# EPICS substitutions: db/elveFlow.substitutions
# asyn record
file "$(ASYN)/db/asynRecord.db"
{
pattern
{ P,	 		    R, 	  PORT,        ADDR, IMAX, OMAX}
{"XF11ID-ES\{elveFlowOB1\}:", asyn, elveFlowOB1, 0,    80,   80}
}
# Analog outputs, analog inputs
file "$(ELVEFLOW)/db/elveFlow.template"
{
pattern
{ P,         R,      		    PORT,        ADDR, DRVL,   DRVH, PREC}
{ XF11ID-ES, "\{elveFlowOB1\}", elveFlowOB1, 0,    0.,     500., 2}
}
